Staubli VAL3: JointState.dtx

public num nSeq
public num nJoints[10]
